FUNCTION_BLOCK Q_FillAttributes (* Command change fill attributes ( Part 6 - F.32 ) *)
  (* Standard: ISO 11783-6; Description: Copyright (c) 2022 HR Agrartechnik GmbH This program and the accompanying materials are made available under the terms of the Eclipse Public License 2.0 which is available at https://www.eclipse.org/legal/epl-2.0/ SPDX-License-Identifier: EPL-2.0 see Description Tab *)
  (* Version 1.0, 2022-07-08, Franz Höpfinger, HR Agrartechnik GmbH *)
  PACKAGE isobus::UT::Q;
  IMPORT eclipse4diac::core::TypeHash;
  IMPORT isobus::UT::Q::IDs::ID_NULL;
  (* Documentation:
  Command change fill attributes ( Part 6 - F.32 )
   This command is used to change the fill attributes in a fill attributes object.
   param[in] {objectID, uint16_t}
   Object ID
   param[in] {fillType, uint8_t}
   New fill type (see Part 6 - B.14.4)
   param[in] {colour, uint8_t}
   New fill colour (see Part 6 - B.14.4)
   param[in] {fillPatternObjectID, uint16_t}
   New fill pattern (see Part 6 - B.14.4)
   Return Values: 
   int16_t
    - VT_E_NO_ERR (0) - OK
   - VT_E_OVERFLOW (-6) - buffer overflow
   - VT_E_NOACT (-8) - Command not possible in current state
   - VT_E_NO_INSTANCE (-21) - No VT client available
   - VT_E_ISO_INSTANCE_INVALID (-129) - Identifier for instance (connection) invalid
   - VT_E_NOT_ALIVE (-130) - Identifier for instance valid, but VT Dead.
  *)
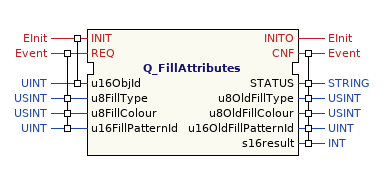
  EVENT_INPUT
    INIT : EInit WITH u16ObjId; (* Service Initialization *)
    REQ WITH u8FillType, u8FillColour, u16FillPatternId; (* Service Request *)
  END_EVENT
  EVENT_OUTPUT
    INITO : EInit; (* Initialization Confirm *)
    CNF WITH STATUS, u16OldFillPatternId, u8OldFillType, u8OldFillColour, s16result; (* Confirmation of Requested Service *)
  END_EVENT
  VAR_INPUT
    u16ObjId : UINT := ID_NULL; (* Object ID *)
    u8FillType : USINT; (* New fill type (see Part 6 - B.14.4) *)
    u8FillColour : USINT; (* New fill colour (see Part 6 - B.14.4) *)
    u16FillPatternId : UINT := ID_NULL; (* New fill pattern (see Part 6 - B.14.4) *)
  END_VAR
  VAR_OUTPUT
    STATUS : STRING; (* Service Status *)
    u8OldFillType : USINT; (* Old fill type (see Part 6 - B.14.4) *)
    u8OldFillColour : USINT; (* Old fill colour (see Part 6 - B.14.4) *)
    u16OldFillPatternId : UINT; (* Old fill pattern (see Part 6 - B.14.4) *)
    s16result : INT; (* retval see description *)
  END_VAR
END_FUNCTION_BLOCK
